// TIA Portal V18 export
VAR_GLOBAL   // PLC tag table "LSql_UserConstants"
END_VAR
VAR_GLOBAL CONSTANT   // user constants
   LSQL_NUMBER_OF_COLUMNS_MAX : UInt := 9;   // upper bound of array for expected columns (zero-based!)
   LSQL_NUMBER_OF_ROWS_MAX : UInt := 9;   // upper bound of array for expected rows (zero-based!)
   LSQL_NUMBER_OF_ROWS_PER_CYCLE : USInt := 0;   // number of rows to be deserialized per cycle (0 = all at once)
END_VAR
